FUNCTION_BLOCK FBMotion
VAR
	AxisPower: MC_Power;
	AxisMoveabsolute: MC_MoveAbsolute;
	AxisHome: MC_Home;
	AxisReset: MC_Reset;
	bHomeExec: BOOL;
	bMoveExec: BOOL;
	MoveToHome: LREAL;
	rVelocity: LREAL := 30;
	rAcceleration: LREAL := 1000;
	rDeceleration: LREAL := 1000;
	rJerk: LREAL := 1000;
	HomeOptions: ST_HomingOptions;
	MoveOptions: ST_MoveOptions;
	PowerOptions: ST_PowerOptions;
	PowerBufferMode: MC_BufferMode;
	HomingMode: MC_HomingMode;
	HomeBufferMode: MC_BufferMode;
	MoveBufferMove: MC_BufferMode;
	MoveBufferMode: MC_BufferMode;
	nDistanceToTarget: INT;
	rDistanceToTarget: LREAL;
	bResetExec: BOOL;
	luku: INT;
END_VAR
VAR_OUTPUT
	bPowerStatus: BOOL;
END_VAR
VAR
	AxisJog: MC_Jog;
	bJogForward: BOOL;
	bJogBackward: BOOL;
	JogMode: E_JogMode := E_JOGMODE.MC_JOGMODE_CONTINOUS;
	rJogVelocity: LREAL := 30;
	rJogAcceleration: LREAL := 1000;
	rJogDeceleration: LREAL := 1000;
	rJogJerk: LREAL := 1000;
	rJogMoveToPos: LREAL;
	rMoveToPos: LREAL;
	eHomeState: E_HomeState;
	bHomeCmd: BOOL;
	tonHomeDelay: TON := (PT := TIME#2S0MS);
	tonSecondDelay: TON := (PT := TIME#500MS);
	tonFinalDelay: TON := (PT := TIME#1S0MS);
	fbSetPosition: MC_SetPosition;
	bSetPosition: BOOL;
	rSetPosition: LREAL := 0;
	SetPos: ST_McOutputs;
END_VAR
VAR_INPUT
	bHomeCalibrationCam: BOOL;
END_VAR
VAR
	bPowerEnable: BOOL := TRUE;
END_VAR
VAR_IN_OUT
	AxisRef: AXIS_REF;
END_VAR
VAR
	MoveOut: ST_McOutputs;
	HomeOut: ST_McOutputs;
	PowerOut: ST_McOutputs;
	JogOut: ST_McOutputs;
	ResetOut: ST_McOutputs;
END_VAR

VAR_OUTPUT
	bHomed: BOOL;
	bP2P_Ready: BOOL;
END_VAR

AxisPower(
	Axis:= AxisRef, 
	Enable:= bPowerEnable, 
	Enable_Positive:= TRUE, 
	Enable_Negative:= TRUE, 
	Override:= 100.0, 
	BufferMode:= PowerBufferMode, 
	Options:= PowerOptions, 
	Status=> bPowerStatus, 		
	Busy=> PowerOut.Busy,        
	Active=> PowerOut.Active,      
	Error=> PowerOut.Error,       
	ErrorID=> PowerOut.ErrorID);    

(*	
AxisHome(
	Axis:= AxisRef, 
	Execute:= bHomeExec, 
	Position:= MoveToHome, 
	HomingMode:= HomingMode, 
	BufferMode:= HomeBufferMode, 
	Options:= HomeOptions, 
	bCalibrationCam:= bHomeCalibrationCam, 
	Done=> 				HomeOut.Done, 
	Busy=> 				HomeOut.Busy, 
	Active=> 			HomeOut.Active, 
	CommandAborted=> 	HomeOut.CommandAborted, 
	Error=> 			HomeOut.Error, 
	ErrorID=> 			HomeOut.ErrorID);
	*)

AxisReset(
	Axis:= AxisRef, 
	Execute:= bResetExec, 
	Done=> ResetOut.Done, 
	Busy=> ResetOut.Busy, 
	Error=> ResetOut.Error, 
	ErrorID=> ResetOut.ErrorID);

//bResetExec := FALSE;
	
AxisMoveabsolute(
	Axis:= AxisRef, 
	Execute:= bMoveExec, 
	Position:= rMoveToPos, 
	Velocity:= rVelocity, 
	Acceleration:= rAcceleration, 
	Deceleration:= rDeceleration, 
	Jerk:= rJerk, 
	BufferMode:= MoveBufferMode, 
	Options:= MoveOptions, 
	Done=> 				MoveOut.Done, 
	Busy=> 				MoveOut.Busy, 
	Active=> 			MoveOut.Active, 
	CommandAborted=> 	MoveOut.CommandAborted, 
	Error=> 			MoveOut.Error, 
	ErrorID=> 			MoveOut.ErrorID);
	
bMoveExec := FALSE;

AxisJog(
	Axis:= AxisRef , 
	JogForward:= bJogForward, 
	JogBackwards:= bJogBackward, 
	Mode:= JogMode, 
	Position:= rJogMoveToPos, 
	Velocity:= rJogVelocity, 
	Acceleration:= rJogAcceleration, 
	Deceleration:= rJogDeceleration, 
	Jerk:= rJogJerk, 
	Done=> JogOut.Done, 
	Busy=> JogOut.Busy, 
	Active=> JogOut.Active, 
	CommandAborted=> JogOut.CommandAborted, 
	Error=> JogOut.Error, 
	ErrorID=> JogOut.ErrorID);

fbSetPosition(
	Axis:= AxisRef, 
	Execute:= bSetPosition, 
	Position:= rSetPosition, 
	Mode:= FALSE, 
	Options:= , 
	Done=> SetPos.Done, 
	Busy=> SetPos.Busy, 
	Error=> SetPos.Error, 
	ErrorID=> SetPos.ErrorID);

tonHomeDelay(IN:= eHomeState = E_HomeState.Delay);
tonSecondDelay(IN:= eHomeState = E_HomeState.SecondDelay);	
tonFinalDelay(IN:= eHomeState = E_HomeState.FinalDelay);		
bHomed := FALSE;



CASE eHomeState OF
	E_HomeState.Inactive:
		 IF bHomeCmd THEN
			 eHomeState := E_HomeState.Jog;
		 END_IF
	E_HomeState.Jog:
		bJogBackward:=TRUE;
		IF bHomeCalibrationCam THEN
			bJogBackward:=FALSE;
			eHomeState := E_HomeState.Delay;
		END_IF
//	E_HomeState.Delay:
//		 IF tonHomeDelay.Q THEN
//			 eHomeState := E_HomeState.SetPos;
//		 END_IF		
//// homing lisä
	E_HomeState.Delay:
		IF tonHomeDelay.Q THEN
			eHomeState := E_HomeState.SecondPhase;
		END_IF
	E_HomeState.SecondPhase:
		IF bHomeCalibrationCam THEN
			bJogForward:= TRUE;
			eHomeState := E_HomeState.SecondDelay;
		END_IF
	E_HomeState.SecondDelay:
		IF tonSecondDelay.Q THEN
			bJogForward:= FALSE;
			eHomeState := E_HomeState.FinalHoming;
		END_IF
	E_HomeState.FinalHoming:
		rJogVelocity := 2;
		bJogBackward:= TRUE;
		IF bHomeCalibrationCam THEN
			bJogBackward:= FALSE;
			rJogVelocity := 30;
			eHomeState:= E_HomeState.FinalDelay;
		END_IF
	E_HomeState.FinalDelay:
		IF tonFinalDelay.Q THEN
			eHomeState := E_HomeState.SetPos;
		END_IF
////////
	E_HomeState.SetPos:
		bSetPosition := TRUE;
		IF SetPos.Done THEN
			bSetPosition := FALSE;
			eHomeState := E_HomeState.HomedReady;
		END_IF	
	(*
	E_HomeState.P2P:
		P2P(0);
		IF MoveOut.Done THEN
			eHomeState := E_HomeState.HomedReady;
		END_IF
	*)
	E_HomeState.HomedReady:
		bHomed := TRUE;
			
END_CASE

 bHomeCmd := FALSE;
 
 rDistanceToTarget := ABS(AxisRef.NcToPlc.ActPos - rMoveToPos);
 bP2P_Ready := rDistanceToTarget < 0.1 AND bHomed;

METHOD FindHome : BOOL
VAR_INPUT
END_VAR
IF eHomeState = E_HomeState.Inactive THEN
	bHomeCmd := TRUE;
	FindHome := TRUE;
ELSE
	FindHome := FALSE;
END_IF
END_METHOD

METHOD P2P : BOOL
VAR_INPUT
	TargetPos: LREAL;
END_VAR


IF bPowerStatus THEN
	rMoveToPos := TargetPos;
	bMoveExec := TRUE;
	P2P := TRUE;
	bP2P_Ready := FALSE;
ELSE
	P2P := FALSE;
END_IF
END_METHOD

METHOD PowerOff : BOOL
VAR_INPUT
END_VAR
bPowerEnable := FALSE;
END_METHOD

METHOD PowerOn : BOOL
VAR_INPUT
END_VAR
bPowerEnable := TRUE;
END_METHOD

METHOD Reset : BOOL
VAR_INPUT
END_VAR
bResetExec := TRUE;
END_METHOD

END_FUNCTION_BLOCK

(* stored: Version 1.1.0.1, ProductVersion 3.1.4024.12
   POU FBMotion: Id {7a5b8d4f-57ac-4dc7-8374-438f1a1cdab8}, SpecialFunc None
   Method FindHome: Id {91988a60-917d-4363-bd4e-8ca6476d9857}
   Method P2P: Id {300f509f-2a8d-42a7-9d6e-2928976bbf3c}
   Method PowerOff: Id {e863b680-91a8-4341-b688-19132c073e0a}
   Method PowerOn: Id {d85ef4ae-a3e4-4526-bc8c-ad1ddf7782a2}
   Method Reset: Id {607a3cf8-213a-4b0f-8ad1-284e7983a098} *)
